PROGRAM PB_ObjectExecution
VAR
END_VAR

Objects.Machine(StartPb      := DigitalInputs.StartPumpPb,
                RunPumpMotor := Objects.HydraulicPumpMotor.RunMotor);

Objects.HydraulicPumpMotor(Running      => DigitalOutputs.HydraulicPumpRunningLamp);

Objects.Safety(EStopHealthy := DigitalInputs.EStopHealthy);

Objects.HmiInterface();

Objects.Logging();

END_PROGRAM

(* stored: Version 1.1.0.1, ProductVersion 3.1.4024.9
   POU PB_ObjectExecution: Id {3d703912-f3fe-4b39-a127-21dab8e6f7dd}, SpecialFunc None *)
